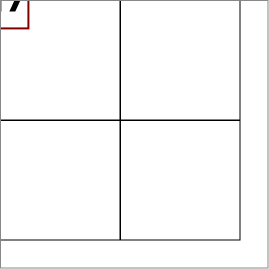
VISUALIZATION V_Control_Xplanar  // 269x269
    Rectangle (0,0 120x120)
    Rectangle (120,0 120x120)
    Rectangle (0,120 120x120)
    Rectangle (120,120 120x120)
    Rectangle (-29,-29 57x57), "M1"
        p3560616238: stMoverVis[1].fPosition_X/2
        p2738717112: (480-stMoverVis[1].fPosition_Y)/2
        p2858320360: stMoverVis[1].fPosition_C
    Rectangle (-29,-29 58x58), "1", invisible if: NOT stStationVis[1].bInit
        p3560616238: stStationVis[1].fPosition_X/2
        p2738717112: (480-stStationVis[1].fPosition_Y)/2
    Rectangle (-29,-29 58x58), "2", invisible if: NOT stStationVis[2].bInit
        p3560616238: stStationVis[2].fPosition_X/2
        p2738717112: (480-stStationVis[2].fPosition_Y)/2
    Rectangle (-29,-29 58x58), "3", invisible if: NOT stStationVis[1].bInit
        p3560616238: stStationVis[3].fPosition_X/2
        p2738717112: (480-stStationVis[3].fPosition_Y)/2
    Rectangle (-29,-29 57x57), "M6"
        p3560616238: stMoverVis[6].fPosition_X/2
        p2738717112: (480-stMoverVis[6].fPosition_Y)/2
        p2858320360: stMoverVis[6].fPosition_C
    Rectangle (-29,-29 57x57), "M5"
        p3560616238: stMoverVis[5].fPosition_X/2
        p2738717112: (480-stMoverVis[5].fPosition_Y)/2
        p2858320360: stMoverVis[5].fPosition_C
    Rectangle (-29,-29 57x57), "M4"
        p3560616238: stMoverVis[4].fPosition_X/2
        p2738717112: (480-stMoverVis[4].fPosition_Y)/2
        p2858320360: stMoverVis[4].fPosition_C
    Rectangle (-29,-29 57x57), "M3"
        p3560616238: stMoverVis[3].fPosition_X/2
        p2738717112: (480-stMoverVis[3].fPosition_Y)/2
        p2858320360: stMoverVis[3].fPosition_C
    Rectangle (-29,-29 57x57), "M2"
        p3560616238: stMoverVis[2].fPosition_X/2
        p2738717112: (480-stMoverVis[2].fPosition_Y)/2
        p2858320360: stMoverVis[2].fPosition_C
    Rectangle (-29,-29 57x57), "M12"
        p3560616238: stMoverVis[12].fPosition_X/2
        p2738717112: (480-stMoverVis[12].fPosition_Y)/2
        p2858320360: stMoverVis[12].fPosition_C
    Rectangle (-29,-29 57x57), "M11"
        p3560616238: stMoverVis[11].fPosition_X/2
        p2738717112: (480-stMoverVis[11].fPosition_Y)/2
        p2858320360: stMoverVis[11].fPosition_C
    Rectangle (-29,-29 57x57), "M10"
        p3560616238: stMoverVis[10].fPosition_X/2
        p2738717112: (480-stMoverVis[10].fPosition_Y)/2
        p2858320360: stMoverVis[10].fPosition_C
    Rectangle (-29,-29 57x57), "M9"
        p3560616238: stMoverVis[9].fPosition_X/2
        p2738717112: (480-stMoverVis[9].fPosition_Y)/2
        p2858320360: stMoverVis[9].fPosition_C
    Rectangle (-29,-29 57x57), "M8"
        p3560616238: stMoverVis[8].fPosition_X/2
        p2738717112: (480-stMoverVis[8].fPosition_Y)/2
        p2858320360: stMoverVis[8].fPosition_C
    Rectangle (-29,-29 57x57), "M7"
        p3560616238: stMoverVis[7].fPosition_X/2
        p2738717112: (480-stMoverVis[7].fPosition_Y)/2
        p2858320360: stMoverVis[7].fPosition_C
END_VISUALIZATION

(* stored: Version 1.1.0.1, ProductVersion 3.1.4024.12
   Visu V_Control_Xplanar: Id {d43f0dbf-72d8-4254-8a8b-664e09fa767d} *)
